Omron CX-Programmer project NewProject (CX-Programmer 9.73)

# PLC IC_Flashing: CP2E-N N

## Global symbols (name address type ; comment)
0.06 BOOL  ; SENSOR M HOME1
A202.07 BOOL  ; Port Enable
A448.00 BOOL  ; Sensor 1
D100 CHANNEL  ; First Source Word
D200 CHANNEL  ; First Destination word
D300 CHANNEL  ; First Control word
W100.00 BOOL  ; Flag On
MODBUS_TCP _CP2E003_ExecuteModTcpServer
Modbus_TCP _CP2E003_ExecuteModTcpServer

## Program NewProgram1 (cyclic task 0)
Local symbols
P_ON BOOL

### Section Section1

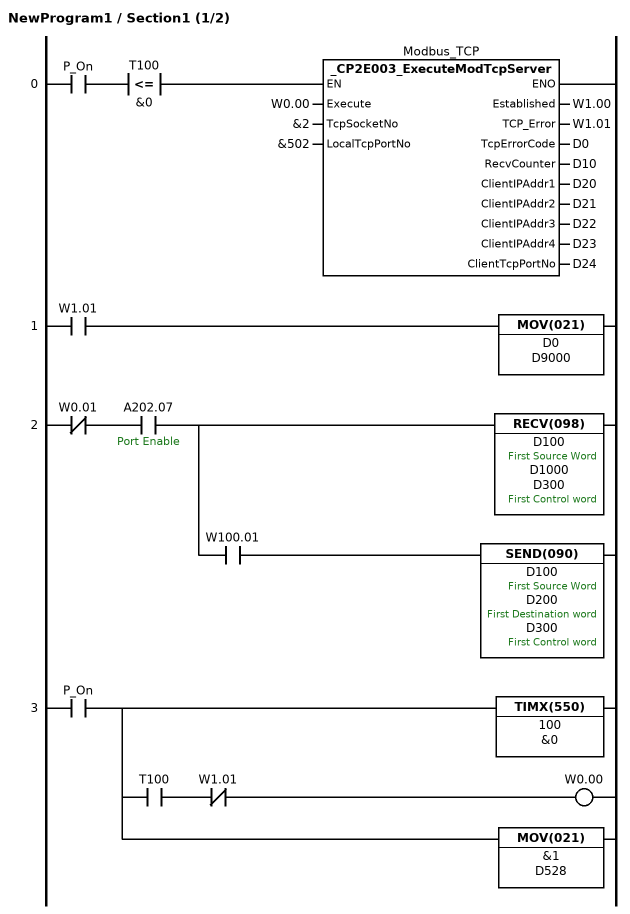
; rung 0
LD P_On
AND<=(315) T100 &0
CALL Modbus_TCP : _CP2E003_ExecuteModTcpServer (Execute := W0.00, TcpSocketNo := &2, LocalTcpPortNo := &502, Established => W1.00, TCP_Error => W1.01, TcpErrorCode => D0, RecvCounter => D10, ClientIPAddr1 => D20, ClientIPAddr2 => D21, ClientIPAddr3 => D22, ClientIPAddr4 => D23, ClientTcpPortNo => D24)
; rung 1
LD W1.01
MOV(021) D0 D9000
; rung 2
LDNOT W0.01
AND A202.07  ; Port Enable
RECV(098) D100 D1000 D300  ; First Source Word, First Control word
AND W100.01
SEND(090) D100 D200 D300  ; First Source Word, First Destination word, First Control word
; rung 3
LD P_On
OUT TR0
TIMX(550) 100 &0
AND T100
ANDNOT W1.01
OUT W0.00
LD TR0
MOV(021) &1 D528

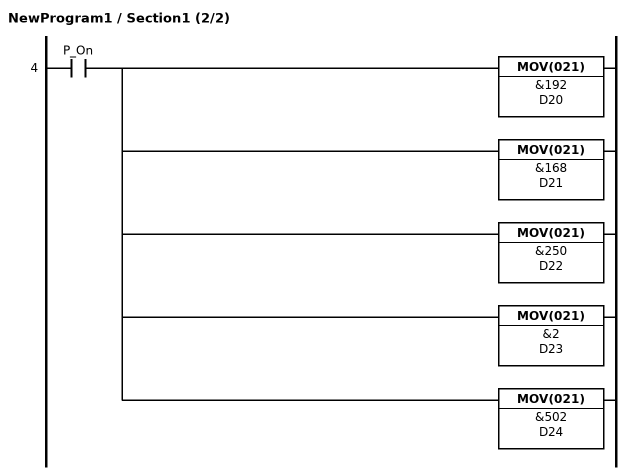
; rung 4
LD P_On
MOV(021) &192 D20
MOV(021) &168 D21
MOV(021) &250 D22
MOV(021) &2 D23
MOV(021) &502 D24

### Section END
; rung 0
END(001)

## Function block _CP2E003_ExecuteModTcpServer (Omron library block, body left out)